PROGRAM MAIN
VAR
    fbEdgeDetection : FB_AuFlankenauswertung;
END_VAR

fbEdgeDetection(Ix_Reset := NOT GVL_CouplerOnDesk.bSelectorSwitchLeftNC);

END_PROGRAM

(* stored: Version 1.1.0.1
   POU MAIN: Id {57926717-fe8b-433d-8dcb-c8a294a9edad}, SpecialFunc None *)
